ABB RAPID module: mfc_MyProduct_path1.mod

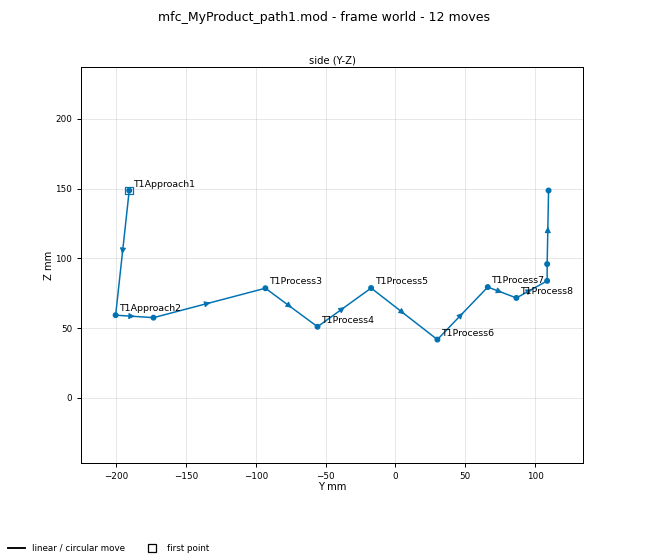
[picture p0: tool path of mfc_MyProduct_path1.mod in frame world, 12 of 12 moves have a stored position in this frame; points joined in program order, loops and branches not executed]
%%%
  VERSION: 1
  LANGUAGE: ENGLISH
%%%

MODULE mfc_MyProduct_path1

!This module is generated by RobotWare Machining FC V3.000. DO NOT EDIT.
!Any changes to this module will be lost when the RW Machining FC application is re-run and the program is exported.
LOCAL VAR robtarget T1Approach1 := [[517.45,-190.77,148.56],[0.0125613,0.79511,-0.606334,0.00099405],[-1,-1,-2,0],[9E+09,9E+09,9E+09,9E+09,9E+09,9E+09]];
LOCAL VAR robtarget T1Approach2 := [[517.45,-200.51,59.24],[0.0125787,0.795105,-0.606341,0.000969681],[-1,-1,-2,0],[9E+09,9E+09,9E+09,9E+09,9E+09,9E+09]];
LOCAL VAR robtarget T1Approach3 := [[517.45,-173.39,57.46],[0.0125744,0.795101,-0.606346,0.000975276],[-1,-1,-2,0],[9E+09,9E+09,9E+09,9E+09,9E+09,9E+09]];
LOCAL VAR robtarget T1Process1  := [[517.45,-143.89,78.49],[0.0125717,0.795104,-0.606342,0.000985399],[-1,-1,-2,0],[9E+09,9E+09,9E+09,9E+09,9E+09,9E+09]];
LOCAL VAR robtarget T1Process2  := [[517.46,-117.6,64.78],[0.0125629,0.795099,-0.606348,0.000998983],[-1,-1,-2,0],[9E+09,9E+09,9E+09,9E+09,9E+09,9E+09]];
LOCAL VAR robtarget T1Process3  := [[517.48,-93.2,78.54],[0.0125443,0.795109,-0.606336,0.00103087],[-1,-1,-2,0],[9E+09,9E+09,9E+09,9E+09,9E+09,9E+09]];
LOCAL VAR robtarget T1Process4  := [[517.47,-55.86,50.95],[0.0125447,0.795105,-0.606342,0.00102],[-1,-1,-2,0],[9E+09,9E+09,9E+09,9E+09,9E+09,9E+09]];
LOCAL VAR robtarget T1Process5  := [[517.45,-17.45,78.67],[0.0125569,0.795093,-0.606356,0.000999938],[-1,-1,-2,0],[9E+09,9E+09,9E+09,9E+09,9E+09,9E+09]];
LOCAL VAR robtarget T1Process6  := [[517.46,30.03,41.75],[0.01256,0.795095,-0.606354,0.00100015],[0,-1,-2,0],[9E+09,9E+09,9E+09,9E+09,9E+09,9E+09]];
LOCAL VAR robtarget T1Process7  := [[517.49,66.12,79.38],[0.0125173,0.795088,-0.606363,0.0010443],[0,-1,-2,0],[9E+09,9E+09,9E+09,9E+09,9E+09,9E+09]];
LOCAL VAR robtarget T1Process8  := [[517.52,86.63,71.6],[0.0124782,0.795095,-0.606355,0.00107598],[0,-1,-2,0],[9E+09,9E+09,9E+09,9E+09,9E+09,9E+09]];
LOCAL VAR robtarget T1Process9  := [[517.54,108.69,83.84],[0.0124477,0.795102,-0.606347,0.00110691],[0,-1,-2,0],[9E+09,9E+09,9E+09,9E+09,9E+09,9E+09]];
LOCAL VAR robtarget T1Withdraw1 := [[517.51,108.68,95.85],[0.0124978,0.795104,-0.606343,0.00106067],[0,-1,-2,0],[9E+09,9E+09,9E+09,9E+09,9E+09,9E+09]];
LOCAL VAR robtarget T1Withdraw2 := [[517.45,109.69,148.56],[0.0125835,0.795103,-0.606343,0.000982652],[0,-1,-2,0],[9E+09,9E+09,9E+09,9E+09,9E+09,9E+09]];
LOCAL VAR num n1ForceX := 0;
LOCAL VAR num n1ForceY := 0;
LOCAL VAR num n1ForceZ := -10;


PROC run_MyProduct_path1 (bool bRecover, bool bSpindleOn)
	FCDeact;

	IF bRecover = true THEN
		FCCalib  mfcTool1_LD \Recovery;
	ELSE
		FCCalib  mfcTool1_LD;
	ENDIF

	IF bSpindleOn = true THEN
		SpindleOn;
	ENDIF

	MoveL T1Approach1, v50, z1,mfcTool1\wobj :=wobj0;
	MoveL T1Approach2, v50, z1,mfcTool1\wobj :=wobj0;
	MoveL T1Approach3, v50, fine,mfcTool1\wobj :=wobj0;

	FCPress1LStart T1Process1, v50 \Fx:= n1ForceX \Fy:= n1ForceY \Fz:= n1ForceZ,50 \ForceFrameRef:=FC_REFFRAME_TOOL \ForceChange:=50 \DampingTune:=100 \TimeOut:=5, \UseSpdFFW, \PosSupvDist:=9e9, fine, mfcTool1 \wobj:=wobj0;
	FCPressL T1Process3, v50, 15, fine, mfcTool1, \wobj:=wobj0;
	FCPressL T1Process4, v50, 15, fine, mfcTool1, \wobj:=wobj0;
	FCPressL T1Process5, v50, 15, fine, mfcTool1, \wobj:=wobj0;
	FCPressL T1Process6, v50, 15, fine, mfcTool1, \wobj:=wobj0;
	FCPressL T1Process7, v50, 15, fine, mfcTool1, \wobj:=wobj0;
	FCPressL T1Process8, v50, 15, fine, mfcTool1, \wobj:=wobj0;
	FCPressL T1Process9, v50, 15, fine, mfcTool1, \wobj:=wobj0;

	FCPressLEnd T1Withdraw1,v50,\ForceChange :=50,\ZeroContactValue := 5;
	MoveL T1Withdraw2, v50, z1,mfcTool1\wobj :=wobj0;

	IF bSpindleOn = true THEN
		SpindleOff;
	ENDIF

ENDPROC

ENDMODULE
